FUNCTION_BLOCK ha_otherthing
  (* Standard: 61499-2 *)
  (* Version 0.1, 2017-00-25, hpea485, UOA *)
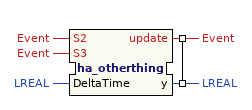
  EVENT_INPUT
    S2;
    S3;
  END_EVENT
  EVENT_OUTPUT
    update WITH y;
  END_EVENT
  VAR_INPUT
    DeltaTime : LREAL := 0.01;
  END_VAR
  VAR_OUTPUT
    y : LREAL;
  END_VAR
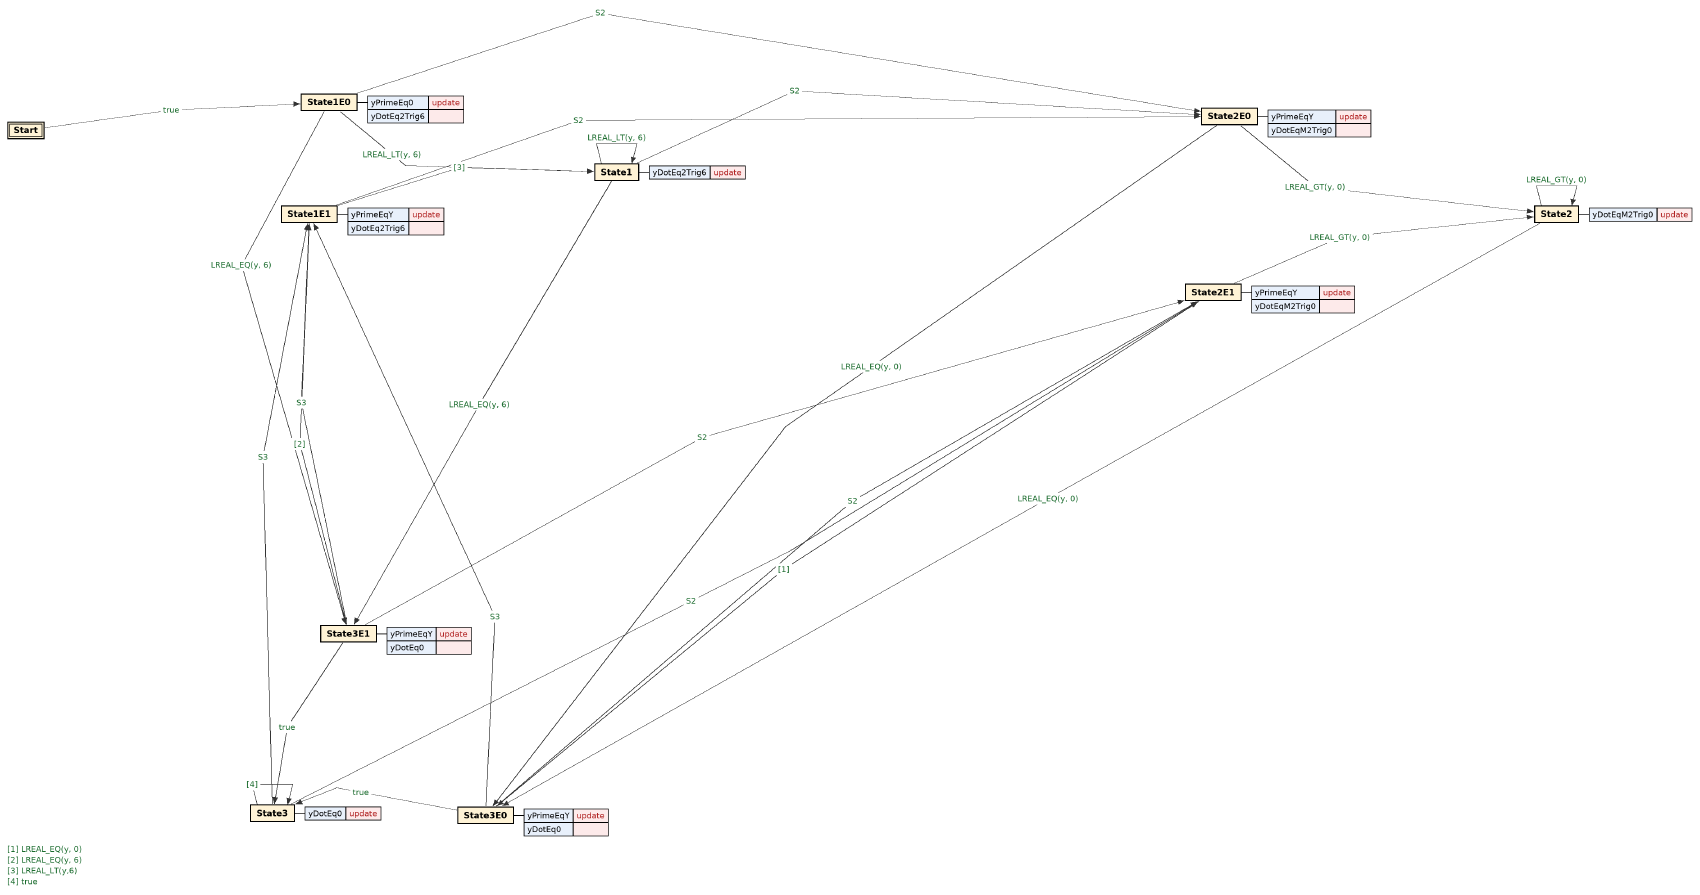
  EC_STATES
    Start;
    State1E0 : yPrimeEq0 -> update, yDotEq2Trig6;
    State1 : yDotEq2Trig6 -> update;
    State2E0 : yPrimeEqY -> update, yDotEqM2Trig0;
    State2E1 : yPrimeEqY -> update, yDotEqM2Trig0;
    State2 : yDotEqM2Trig0 -> update;
    State3E0 : yPrimeEqY -> update, yDotEq0;
    State3E1 : yPrimeEqY -> update, yDotEq0;
    State3 : yDotEq0 -> update;
    State1E1 : yPrimeEqY -> update, yDotEq2Trig6;
  END_STATES
  EC_TRANSITIONS
    Start TO State1E0 := true;
    State1E0 TO State2E0 := S2;
    State1E0 TO State3E1 := LREAL_EQ(y, 6);
    State1E0 TO State1 := LREAL_LT(y, 6);
    State1 TO State2E0 := S2;
    State1 TO State3E1 := LREAL_EQ(y, 6);
    State1 TO State1 := LREAL_LT(y, 6);
    State2E0 TO State3E0 := LREAL_EQ(y, 0);
    State2E0 TO State2 := LREAL_GT(y, 0);
    State2E1 TO State3E0 := LREAL_EQ(y, 0);
    State2E1 TO State2 := LREAL_GT(y, 0);
    State2 TO State3E0 := LREAL_EQ(y, 0);
    State2 TO State2 := LREAL_GT(y, 0);
    State3E0 TO State2E1 := S2;
    State3E0 TO State1E1 := S3;
    State3E0 TO State3 := true;
    State3E1 TO State2E1 := S2;
    State3E1 TO State1E1 := S3;
    State3E1 TO State3 := true;
    State3 TO State2E1 := S2;
    State3 TO State1E1 := S3;
    State3 TO State3 := true;
    State1E1 TO State2E0 := S2;
    State1E1 TO State3E1 := LREAL_EQ(y, 6);
    State1E1 TO State1 := LREAL_LT(y,6);
  END_TRANSITIONS
  ALGORITHM yPrimeEq0 IN C: (* ODE_init *)
y_prime = 0;
  END_ALGORITHM
  ALGORITHM yPrimeEqY IN C: (* ODE_init *)
y_prime = y;
  END_ALGORITHM
  ALGORITHM yDotEq2Trig6 IN C: (* ODE *)
y_dot = 2;
y_trigger = 6;
  END_ALGORITHM
  ALGORITHM yDotEqM2Trig0 IN C: (* ODE *)
y_dot = -2;
y_trigger = 0;
  END_ALGORITHM
  ALGORITHM yDotEq0 IN C: (* ODE *)
y_dot = 0;
  END_ALGORITHM
END_FUNCTION_BLOCK
